{attribute addProperty BoxType "EP2339-0021-0016"}
{attribute addProperty Id "AoeNetIdAT %I*AMSNETID4860StateAT %I*UINT1620"}
{attribute addProperty CRC "782378116"}
{attribute addProperty SizeInBites "64"}
{attribute addProperty SizeInBytes "8"}
TYPE InfoData_2EA22484 :
STRUCT
	{attribute addProperty Name "AoeNetId"}
	AoeNetId AT %I* : AMSNETID;
	{attribute addProperty Name "State"}
	State AT %I* : UINT;
END_STRUCT
END_TYPE

(* stored: Version 1.2.0.0, ProductVersion 3.1.4024.9
   DUT InfoData_2EA22484: Id {76e6396d-a0f0-44f3-8959-7e15924dda8e} *)
